// TIA Portal V19 export
DATA_BLOCK "iDB_ManageState"   // DB20
{ DB_Accessible_From_OPC_UA := 'FALSE' }
// stored: AutoNumber false, DBAccessibleFromOPCUA false, DBAccessibleFromWebserver false, InstanceOfName FB20_ManageState, InstanceOfType FB
"FB20_ManageState"
   // VAR_INPUT
   //    xGlobalSafety { ExternalAccessible := 'False'; ExternalVisible := 'False'; ExternalWritable := 'False'} : Bool;
   //    xGlobalFault { ExternalAccessible := 'False'; ExternalVisible := 'False'; ExternalWritable := 'False'} : Bool;
   //    xInformation { ExternalAccessible := 'False'; ExternalVisible := 'False'; ExternalWritable := 'False'} : Bool;
   // END_VAR
   // VAR_OUTPUT
   //    nGlobalState { ExternalAccessible := 'False'; ExternalVisible := 'False'; ExternalWritable := 'False'} : Int;
   //    xSafetyState { ExternalAccessible := 'False'; ExternalVisible := 'False'; ExternalWritable := 'False'} : Bool;
   // END_VAR
BEGIN
END_DATA_BLOCK
